{attribute 'qualified_only'}
VAR_GLOBAL
	visValveMaskIdx : INT;
	nValveMask 		: DWORD;
	anValveMask 	: ARRAY [0..GVL_AteqConfig.nMaxProgramsToRun -1] OF DWORD;
END_VAR

(* stored: Version 1.1.0.1
   GVL GVL_visVariableMap: Id {e66e5bb2-e186-0a7a-1eb9-6daef8b222c0} *)
